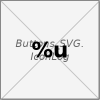
VISUALIZATION ButtonLog  // 100x100
VAR_IN_OUT
	bState : BOOL;
	nNumber : UINT;
	dColor : DWORD;
END_VAR
    Frame (0,0 100x100)
        shows ButtonTemplate(bActive := bState)
    Ellipse (5,5 90x90), colour variable: dColor
    Image (0,0 100x100), image: Buttons_SVG.IconLog
    Textfield (0,0 100x100), "%u", text variable: nNumber
        OnMouseDown: execute { GVL_HMI.fbHMIControl.eScreenRequest := E_BaseVisu.LogView; }
END_VISUALIZATION

(* stored: Version 1.1.0.1, ProductVersion 3.1.4024.11
   Visu ButtonLog: Id {be0113de-8425-4fcf-a286-add62edaa25f} *)
